Fanuc KAREL source: kc00050.KL

-- PROVISIONAL review KL for V1013-1; original PC SHA256 505a2b8f1f730a98cd59f822d39f7bb86360005e28f3d22ad688f85f93d138b2
-- Incomplete behavior may be omitted. Consult companion uncertainty JSON. Do not deploy.
PROGRAM KC00050
%NOLOCKGROUP
BEGIN
  -- UNRESOLVED_PC offsets 5-35; opcodes 27,22,22,1C,22,27,9D,31
  -- UNRESOLVED_PC offsets 40-44; opcodes 7F
END KC00050
